{attribute 'linkalways'} 
{attribute 'no_explicit_call' := 'This FB is a CLASS and must be accessed using methods or properties'}
{attribute 'enable_dynamic_creation'}
FUNCTION_BLOCK FINAL Node_CONCAT EXTENDS Node
VAR
	str1 : _STRING('');
    str2 : _STRING('');
	out : _STRING('');
END_VAR

METHOD PUBLIC  Clone : I_Node
VAR
	pNode : POINTER TO Node_CONCAT;
END_VAR
pNode := __NEW(Node_CONCAT);
Clone := pNode^;
END_METHOD

METHOD FB_init : BOOL
VAR_INPUT
	bInitRetains : BOOL; // if TRUE, the retain variables are initialized (warm start / cold start)
	bInCopyCode : BOOL;  // if TRUE, the instance afterwards gets moved into the copy code (online change)
END_VAR
AddParameter('str1', str1);
AddParameter('str2', str2);
AddOutput('out', out);
END_METHOD

METHOD PROTECTED OnExecute
VAR
END_VAR
out.Value := CONCAT(str1.Value, str2.Value);
END_METHOD

END_FUNCTION_BLOCK

(* stored: Version 1.1.0.1, ProductVersion 3.1.4026.18
   POU Node_CONCAT: Id {ef7f9083-5304-0745-13c5-98adfde0bd94}, SpecialFunc None
   Folder Constructor: Id {94e7cc8d-54e3-065f-0134-75873439a066}
   Method Clone: Id {a666624c-e12e-0bc7-02b6-410f3709226c}
   Method FB_init: Id {f2fd5c95-39d1-0c80-03fc-1ab3dec5594d}
   Method OnExecute: Id {ce41925c-f816-0a05-04e9-66b2280415aa} *)
